// TIA Portal V20 export
DATA_BLOCK "instGetIdentRf"   // DB217
// stored: InstanceOfName GetIdentRf, InstanceOfType FB
"GetIdentRf"
   // VAR_INPUT
   //    identRfAllUnits { ExternalAccessible := 'False'; ExternalVisible := 'False'; ExternalWritable := 'False'} : Array[1.."NO_OF_UNITS"] of "typeEMIdentRf";
   //    numberOfRfReaders : USInt;
   // END_VAR
   // VAR_OUTPUT
   //    selectedUnit : USInt;
   //    selectedEM : USInt;
   //    error : Word;
   // END_VAR
   // VAR_IN_OUT
   //    IdentRfInterfaceHmi : "typeIdentRfHmi";
   // END_VAR
   // VAR
   //    statSelectedEMIdentRf : USInt;
   //    statSelectedUnitIdentRf : USInt;
   // END_VAR
BEGIN
END_DATA_BLOCK
